// TIA Portal V17 export
// export: Created 2023-05-07T12:12:22.2902351Z, ExportSetting WithDefaults, DisplayName Totally Integrated Automation Portal, DisplayVersion V17, DisplayName TIA Portal Openness, DisplayVersion V17, DisplayName TIA Portal Version Control Interface, DisplayVersion V17, DisplayName TIA Portal Test Suite Advanced, DisplayVersion V17, DisplayName STEP 7 Professional, DisplayVersion V17, DisplayName SIMATIC Energy Suite, DisplayVersion V17, DisplayName STEP 7 Safety, DisplayVersion V17, DisplayName WinCC Professional, DisplayVersion V17
DATA_BLOCK "RAMP_DB"   // DB6
VERSION : 0.1
// stored: AutoNumber true, InstanceOfName RAMP, InstanceOfType FB
"RAMP"
   // VAR_INPUT
   //    SetPoint : Real;
   //    Rate : Real;
   //    Reset : Bool;
   // END_VAR
   // VAR_OUTPUT
   //    OUT : Real;
   // END_VAR
   // VAR
   //    TON_1 { ExternalAccessible := 'False'; ExternalVisible := 'False'; ExternalWritable := 'False'} : TON_TIME;
   //    RateDIV : Real;
   //    Q : Bool;
   // END_VAR
BEGIN
END_DATA_BLOCK
